TYPE U_Convert_USINT :
UNION
	nValue		:USINT;					// Unsigned short integer value representation of data
    byValue 	:BYTE;					// Byte value representation of data
	//arrBit		:ARRAY[0..7]OF bool;	   // Bit representation of data
END_UNION
END_TYPE

(* stored: Version 1.1.0.1, ProductVersion 3.1.4024.12
   DUT U_Convert_USINT: Id {23a61af4-fe8e-4b55-8b87-56aabd956e3a} *)
